// TIA Portal V19 export
DATA_BLOCK "Boiler 1"   // DB11
// stored: InstanceOfName Boiler Alarm, InstanceOfType FB
"Boiler Alarm"
   // VAR_INPUT
   //    "Alarm Bit" : Bool;
   // END_VAR
   // VAR
   //    Boiler : Program_Alarm;
   // END_VAR
BEGIN
END_DATA_BLOCK
